PROGRAM MAIN
VAR
	//fbfilesource                                    : FB_VN_FileSourceControl;	
	CAMERA 											: FB_VN_FileSourceControl;	
	raw_image										: ITcVnImage;	
	WORKED_image										: ITcVnImage;	
	ipImageIn              						    :   ITcVnImage;
	display_raw_image								: ITcVnDisplayableImage;		
	
	ipcontours										: ITcVnContainer;	
	number_of_elements								: ULINT;	
	hr 												: HRESULT;	
	cState 											: ETcVnCameraState;	
	green_color										: TcVnVector4_LREAL := [0,255,0,0];	
	Bcolor										: TcVnVector4_LREAL := [100,0,0,0];
	stext											: STRING;
	
	
//	raw_image           :    ITcVnImage;

// QR Code
ipCodeDecodedList   :    ITcVnContainer; 
ipCodeContourList   :    ITcVnContainer;
sCodeAsString       :    STRING(255);

// Watchdog
hrWD                :    HRESULT;
tStop               :    DINT := 20000;
tRest               :    DINT;

// Output
//sText               :    STRING;

// Color
aColorRed           :    TcVnVector4_LREAL := [255, 0, 0];
END_VAR



cState 				:= CAMERA.GetState();

CASE cState OF
	

TCVN_CS_INITIAL, TCVN_CS_OPENING, TCVN_CS_OPENED, TCVN_CS_STARTACQUISITION :

 	hr  := CAMERA.StartAcquisition();  // start Camera acquisition



TCVN_CS_ACQUIRING:
	HR := CAMERA.GetCurrentImage(raw_image);   //get image from file source 
	ipImageIn := raw_image;   //get image from file source 
	
	 IF SUCCEEDED(HR) AND ipImageIn <> 0 THEN
		

		(*hr := F_VN_ConvertColorSpace(raw_image, worked_image, TCVN_CST_RGB_TO_GRAY, hr);
		hr := F_VN_FindContours(worked_image, ipcontours, hr);
		hr := F_VN_GetNumberOfElements(ipcontours,number_of_elements, hr);
		hr := F_VN_DrawContours(ipcontours,-1,raw_image,green_color,2, hr);
		
		stext := ULINT_TO_STRING(number_of_elements);
		
		hr := F_VN_PutText(STEXT, raw_image, 70,270,TCVN_FT_HERSHEY_COMPLEX,2 , Bcolor, hr);
		
	END_IF

		hr :=  F_VN_CopyIntoDisplayableImage(raw_image, display_raw_image, hr); *)
	
 		
		
 	//QRCODE();
	Barcode();
END_IF	
TCVN_CS_ERROR:	

	hr 	:= CAMERA.Reset();
END_CASE

END_PROGRAM

(* stored: Version 1.1.0.1, ProductVersion 3.1.4024.12
   POU MAIN: Id {7baf06ec-f7b0-4131-a547-bb69c3d04e8e}, SpecialFunc None *)
